FUNCTION_BLOCK Skill_PickPlace EXTENDS FB_Template_Skill
VAR_INPUT
	Rob: POINTER TO FB_ROB_MANIP;
	sPickReference: STRING;
END_VAR
VAR_OUTPUT
	
END_VAR
VAR
	
END_VAR

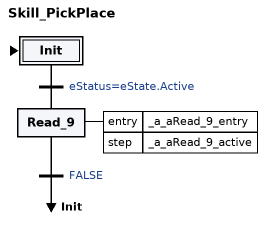
INITIAL_STEP Init:
END_STEP
TRANSITION FROM Init TO Read_9
    := eStatus=eState.Active;
END_TRANSITION
STEP Read_9:
    _a_aRead_9_entry(P1);  // entry action
    _a_aRead_9_active(N);  // step action
END_STEP
TRANSITION FROM Read_9 TO Init
    := FALSE;
END_TRANSITION

ACTION _a_aRead_9_active:

END_ACTION

ACTION _a_aRead_9_entry:

END_ACTION

END_FUNCTION_BLOCK

(* stored: Version 1.1.0.1, ProductVersion 3.1.4026.18
   POU Skill_PickPlace: Id {0265789f-44be-4ed2-bfd3-e8ebd7334e24}, SpecialFunc None
   Action _a_aRead_9_active: Id {0ed342dc-ab1a-41b5-b1e5-c1ad080eceec}
   Action _a_aRead_9_entry: Id {8e8ec55a-a4d1-45bf-9399-57ef58eac1be} *)
